INTERFACE I_CylinderMover EXTENDS ITaskStatus

METHOD PUBLIC MoveToTarget : BOOL
VAR_INPUT
END_VAR
END_METHOD

END_INTERFACE

(* stored: Version 1.1.0.1, ProductVersion 3.1.4024.4
   Itf I_CylinderMover: Id {dc15a651-b873-4ae0-ba7e-14d24bed9057}
   Method MoveToTarget: Id {f95a03fa-34d3-4a81-91b8-5221977815de} *)
